IF Device.DSo.Node=0 THEN Get_Node(); END_IF
_w1 := NOT (Device.DSo.Node=0);
IF _w1 THEN Get_State(); END_IF
IF _w1 AND (Device.CanOpen.Device_State=_3SCOS.DED.DEVICE_STATE.CONFIGURED) THEN State_PreOp(); END_IF
_w2 := True;
IF _w2 THEN PDO_Units(); END_IF
IF _w2 THEN Process_Alarms(); END_IF
_w3 := Device.CanOpen.Device_State=_3SCOS.DED.DEVICE_STATE.RUNNING;
IF _w3 THEN Write_SDO(); END_IF
IF _w3 AND Device.CanOpen.Read_Once THEN Read_SDO(); END_IF
_w4 := Device.CanOpen.Device_State=_3SCOS.DED.DEVICE_STATE.RUNNING;
IF _w4 THEN
    SDO_CLK(PT := t#500ms); // Burkert_OSCAT_BASIC.CLK_PRG
END_IF
IF _w4 THEN
    AutoRead_CLK(PT := T#30s); // Burkert_OSCAT_BASIC.CLK_PRG
END_IF
IF AutoRead_CLK.Q THEN _w5 := True; END_IF
Device.CanOpen.Read_Once := _w5;
Device.PDO.NamurStatus.eNamur := SEL(Device.CanOpen.Device_State=_3SCOS.DED.DEVICE_STATE.RUNNING, eNamur107.Offline, Device.PDO.NamurStatus.eNamur);

END_FUNCTION_BLOCK

// Level_1_Devices/Burkert Library/CanOpen/CanOpen_8228
FUNCTION_BLOCK CanOpen_8228
VAR_INPUT
	Device: 	REFERENCE TO cCanOpen_8228;
	CanOpen:	REFERENCE TO _3SCOS.CANRemoteDevice_Diag;
	Conductivity_Units:eUnits:=eUnits.uS_cm;
	Temperature_Units:eUnits:=eUnits.C;
END_VAR
VAR_OUTPUT
END_VAR
VAR
	Concentration_Alarm:Burkert.Analog_Alarm_UDFB;
	Conductivity_Alarm:Burkert.Analog_Alarm_UDFB;
	Resistivity_Alarm:Burkert.Analog_Alarm_UDFB;
	TDS_Alarm:Burkert.Analog_Alarm_UDFB;
	Temp_Alarm:Burkert.Analog_Alarm_UDFB;
	
	Write_Data:Bytes_Dword;
	SDO_CLK:Burkert_OSCAT_BASIC.CLK_PRG;
	AutoRead_CLK:Burkert_OSCAT_BASIC.CLK_PRG;
	SDO_Read:CIA405.SDO_READ4;
	SDO_Write:CIA405.SDO_WRITE_DATA;

	
	
END_VAR

CanOpen_NMT();
IF Device.CanOpen.Device_State=_3SCOS.DED.DEVICE_STATE.RUNNING THEN
	AutoRead_CLK(PT:=T#60S);
	SDO_CLK(PT:=T#200MS);

	Alarms();
	IF Device.CanOpen.Read_Once THEN
		READ_SDO();
	ELSE
		Write_SDO();
	END_IF
END_IF

IF AutoRead_CLK.Q THEN
	Device.CanOpen.Read_Once:=TRUE;
END_IF
Translate();
Units();
Alarms();

Device.Ready:=(Device.Namur<2);
Device.TDS.Ready:=FPU.IsRealNumber(f:=Device.TDS.EU) AND Device.Namur<>0;
Device.Concentration.Ready:=FPU.IsRealNumber(f:=Device.Concentration.EU) AND Device.Namur<>0;
Device.Conductivity.Ready:=FPU.IsRealNumber(f:=Device.Conductivity.EU) AND Device.Namur<>0;
Device.Resistivity.Ready:=FPU.IsRealNumber(f:=Device.Resistivity.EU) AND Device.Namur<>0;
Device.Temperature.Ready:=FPU.IsRealNumber(f:=Device.Temperature.EU) AND Device.Namur<>0;

Device.DSO.StrNamur:=TO_STRING(Device.DSO.NamurNe107.eNamur);

END_FUNCTION_BLOCK

// Level_1_Devices/Burkert Library/CanOpen/CanOpen_8691
FUNCTION_BLOCK CanOpen_8691
VAR_INPUT

	LOCKOUT:BOOL;
	//Online:BOOL;
	Interlock:BOOL;
	Error_Delay_S:INT:=10;
	CanOpen:	REFERENCE TO _3SCOS.CANRemoteDevice_Diag;
	
	
	
END_VAR
VAR_OUTPUT
	Status	:INT;
	Output	:REAL;
END_VAR
VAR_IN_OUT
	Device	:cCanOpen_8691;
END_VAR
VAR

	TON_1: TON;
	TOF_0: TOF;
	R_TRIG_0: R_Trig;
	F_TRIG_0: F_Trig;

	SDO_CLK:Burkert_OSCAT_BASIC.CLK_PRG;
	AutoRead_CLK:Burkert_OSCAT_BASIC.CLK_PRG;
	SDO_Read:CIA405.SDO_READ4;
	SDO_Write:CIA405.SDO_WRITE_DATA;
	Basic_BCV:Basic_BCV_UDFB;
	
	
	CanRestart:TON;
	SetCommunicationState:_3SCOS.DED.ERROR;



END_VAR

(* body of a kind this reader does not render *)

END_FUNCTION_BLOCK

// Level_1_Devices/Burkert Library/CanOpen/CanOpen_8694
FUNCTION_BLOCK CanOpen_8694
VAR_INPUT
	CutOff:REAL:=0;
	LockOut_NC:BOOL:=TRUE;
	Permissive_NC:BOOL:=TRUE;
	Error_PCT:REAL:=10;
	Error_Delay_S:INT:=10;
	CanOpen:	REFERENCE TO _3SCOS.CANRemoteDevice_Diag;
	Device	:	REFERENCE TO cCanOpen_8694;
	
	
	
END_VAR
VAR_OUTPUT
	Status	:INT;
	Output	:REAL;
END_VAR
VAR_IN_OUT
	
END_VAR
VAR

	CanRestart:TON;

	Status_CLK:Burkert_OSCAT_BASIC.CLK_PRG;
	SDO_CLK:Burkert_OSCAT_BASIC.CLK_PRG;
	AutoRead_CLK:Burkert_OSCAT_BASIC.CLK_PRG;
	GetState_CLK:Burkert_OSCAT_BASIC.GEN_PULSE;
	SDO_Read:CIA405.SDO_READ4;
	SDO_Write:CIA405.SDO_WRITE_DATA;
	SDO_Data:ARRAY[1..4] OF BYTE;
	Write_Data:Bytes_Dword;
	
	
	Base_ACV:Basic_ACV_UDFB;
	
	SetCommunicationState:_3SCOS.DED.ERROR;
	//deiInfo:_3SCOS.DED.DEVICE_INFO;
	GetState:			CIA405.GET_STATE;
	CIA_State:			CIA405.DEVICE_STATE;
	NMT:				CIA405.NMT;
	CanState:			_3SCOS.DED.DEVICE_STATE;
	Device_State:		_3SCOS.DED.DEVICE_STATE;
	GetState_eError:	_3SCOS.DED.ERROR;
	Start_Available:BOOL;
	Ref_OK:Bool;
END_VAR

(* body of a kind this reader does not render *)

END_FUNCTION_BLOCK

// Level_1_Devices/Burkert Library/CanOpen/CanOpen_MS02
FUNCTION_BLOCK CanOpen_MS02
VAR_INPUT
	CanOpen:	REFERENCE TO _3SCOS.CANRemoteDevice_Diag;
	
END_VAR
VAR_OUTPUT
END_VAR
VAR
	SDO_CLK:Burkert_OSCAT_BASIC.CLK_PRG;
	AutoRead_CLK:Burkert_OSCAT_BASIC.CLK_PRG;
	SDO_Read:CIA405.SDO_READ4;
	SDO_Write:CIA405.SDO_WRITE_DATA;
	ALARM_0: Burkert.Analog_Alarm_UDFB;
	ALARM_1: Burkert.Analog_Alarm_UDFB;
	
END_VAR
VAR_IN_OUT
	Sensor: cCanOpen_MS02;
	
END_VAR

CanOpen_NMT();
IF Sensor.CanOpen.Device_State=_3SCOS.DED.DEVICE_STATE.RUNNING THEN
	AutoRead_CLK(PT:=T#60S);
	SDO_CLK(PT:=T#200MS);

	Alarms();
	IF Sensor.CanOpen.Read_Once THEN
		READ_SDO();
	ELSE
		Write_SDO();
	END_IF
END_IF

IF AutoRead_CLK.Q THEN
	Sensor.CanOpen.Read_Once:=TRUE;
END_IF

END_FUNCTION_BLOCK

// Level_1_Devices/Burkert Library/CanOpen/CanOpen_MS03
FUNCTION_BLOCK CanOpen_MS03
VAR_INPUT
	CanOpen:	REFERENCE TO _3SCOS.CANRemoteDevice_Diag;
	
END_VAR
VAR_OUTPUT
END_VAR
VAR
	SDO_CLK:Burkert_OSCAT_BASIC.CLK_PRG;
	AutoRead_CLK:Burkert_OSCAT_BASIC.CLK_PRG;
	SDO_Read:CIA405.SDO_READ4;
	SDO_Write:CIA405.SDO_WRITE_DATA;
	ALARM_0: Burkert.Analog_Alarm_UDFB;
	ALARM_1: Burkert.Analog_Alarm_UDFB;
	
END_VAR
VAR_IN_OUT
	Sensor: cCanOpen_MS03;
	
END_VAR

CanOpen_NMT();
IF Sensor.CanOpen.Device_State=_3SCOS.DED.DEVICE_STATE.RUNNING THEN
	AutoRead_CLK(PT:=T#60S);
	SDO_CLK(PT:=T#200MS);

	Alarms();
	IF Sensor.CanOpen.Read_Once THEN
		READ_SDO();
	ELSE
		Write_SDO();
	END_IF
END_IF

IF AutoRead_CLK.Q THEN
	Sensor.CanOpen.Read_Once:=TRUE;
END_IF

END_FUNCTION_BLOCK

// Level_1_Devices/Burkert Library/CanOpen/CanOpen_MS04
FUNCTION_BLOCK CanOpen_MS04
VAR_INPUT
	CanOpen:	REFERENCE TO _3SCOS.CANRemoteDevice_Diag;
	
END_VAR
VAR_OUTPUT
END_VAR
VAR
	SDO_CLK:Burkert_OSCAT_BASIC.CLK_PRG;
	AutoRead_CLK:Burkert_OSCAT_BASIC.CLK_PRG;
	SDO_Read:CIA405.SDO_READ4;
	SDO_Write:CIA405.SDO_WRITE_DATA;
	ALARM_0: Burkert.Analog_Alarm_UDFB;
	ALARM_1: Burkert.Analog_Alarm_UDFB;
	
END_VAR
VAR_IN_OUT
	Sensor: cCanOpen_MS04;
	
END_VAR

CanOpen_NMT();
IF Sensor.CanOpen.Device_State=_3SCOS.DED.DEVICE_STATE.RUNNING THEN
	AutoRead_CLK(PT:=T#60S);
	SDO_CLK(PT:=T#200MS);

	Alarms();
	IF Sensor.CanOpen.Read_Once THEN
		READ_SDO();
	ELSE
		Write_SDO();
	END_IF
END_IF

IF AutoRead_CLK.Q THEN
	Sensor.CanOpen.Read_Once:=TRUE;
END_IF

END_FUNCTION_BLOCK

// Level_1_Devices/Burkert Library/CanOpen/CanOpen_MS05
FUNCTION_BLOCK CanOpen_MS05
VAR_INPUT
	CanOpen:	REFERENCE TO _3SCOS.CANRemoteDevice_Diag;
	
END_VAR
VAR_OUTPUT
END_VAR
VAR
	SDO_CLK:Burkert_OSCAT_BASIC.CLK_PRG;
	AutoRead_CLK:Burkert_OSCAT_BASIC.CLK_PRG;
	SDO_Read:CIA405.SDO_READ4;
	SDO_Write:CIA405.SDO_WRITE_DATA;
	ALARM_0: Burkert.Analog_Alarm_UDFB;
	ALARM_1: Burkert.Analog_Alarm_UDFB;
	
END_VAR
VAR_IN_OUT
	Sensor: cCanOpen_MS05;
	
END_VAR

CanOpen_NMT();
IF Sensor.CanOpen.Device_State=_3SCOS.DED.DEVICE_STATE.RUNNING THEN
	AutoRead_CLK(PT:=T#60S);
	SDO_CLK(PT:=T#200MS);

	Alarms();
	IF Sensor.CanOpen.Read_Once THEN
		READ_SDO();
	ELSE
		Write_SDO();
	END_IF
END_IF

IF AutoRead_CLK.Q THEN
	Sensor.CanOpen.Read_Once:=TRUE;
END_IF

END_FUNCTION_BLOCK

// Level_1_Devices/Burkert Library/eDip/eDip_8098_CTRL
FUNCTION_BLOCK eDip_8098_CTRL
VAR_INPUT
	Device: REFERENCE TO ceDip_8098;
	Gateway: REFERENCE TO ME43_SDO;
	Node:Byte;
	Temperature_Units:eUnits:=eUnits.C;
	Flow_Units:eUnits:=eUnits.lpm;
	Volume_Units:eUnits:=eUnits.l;
END_VAR
VAR_OUTPUT
END_VAR
VAR
	Data:Bytes_Dword;
	Alarm:ARRAY[0..5] OF Burkert.Analog_Alarm_UDFB;
	Device_Valid:BOOL;
	Gateway_Valid:BOOL;
	F_trig_0:F_Trig;
	Startup_Ton:Ton;
	
	
END_VAR

Device.DSO.Node:=Node;


Device_Valid:=__ISVALIDREF(Device);
Gateway_Valid:=__ISVALIDREF(Gateway);
Device.DSO.Node:=Node;

IF  Device_Valid  THEN 
	Parse_RX();
END_IF;
StartUp_Ton(In:=Gateway_Valid AND Device_Valid ,PT:=T#1S);

IF Gateway_Valid AND StartUp_Ton.Q THEN
	Process_Alarms();
	Reset_Counters();
	Device.TCP_State:=Gateway.CommState;
	Device.strTCPstate:=TO_STRING(Device.TCP_State);
END_IF

END_FUNCTION_BLOCK

// Level_1_Devices/Burkert Library/eDip/eDip_8228_MEx3
FUNCTION_BLOCK eDip_8228_MEx3
VAR_INPUT
	Device: REFERENCE TO ceDip_8228;
	GW_Connected:BOOL;
	Node:byte;
END_VAR
VAR_OUTPUT
END_VAR
VAR
	data:Bytes_Dword;
	Concentration_Alarm:Burkert.Analog_Alarm_UDFB;
	Conductivity_Alarm:Burkert.Analog_Alarm_UDFB;
	Resistivity_Alarm:Burkert.Analog_Alarm_UDFB;
	TDS_Alarm:Burkert.Analog_Alarm_UDFB;
	Temp_Alarm:Burkert.Analog_Alarm_UDFB;
	Concentration_Native:REAL;
	Conductivity_Native:REAL;
	Resistivity_Native:REAL;
	TDS_Native:REAL;
	Temperature_Native:REAL;
	
	
END_VAR

Device.DSO.Node:=Node;
Translate();
Units();
Alarms();

Device.Ready:=(Device.Namur<2) AND GW_Connected ;
Device.TDS.Ready:=FPU.IsRealNumber(f:=Device.TDS.EU)AND GW_Connected AND Device.Namur<>0;
Device.Concentration.Ready:=FPU.IsRealNumber(f:=Device.Concentration.EU)AND GW_Connected AND Device.Namur<>0;
Device.Conductivity.Ready:=FPU.IsRealNumber(f:=Device.Conductivity.EU)AND GW_Connected AND Device.Namur<>0;
Device.Resistivity.Ready:=FPU.IsRealNumber(f:=Device.Resistivity.EU)AND GW_Connected AND Device.Namur<>0;
Device.Temperature.Ready:=FPU.IsRealNumber(f:=Device.Temperature.EU)AND GW_Connected AND Device.Namur<>0;

END_FUNCTION_BLOCK

// Level_1_Devices/Burkert Library/eDip/eDip_8312
FUNCTION_BLOCK eDip_8312
VAR_INPUT
	Device:REFERENCE TO c8312;
	GW_Connected:BOOL;
	Node:BYTE;
END_VAR
VAR_OUTPUT
END_VAR
VAR
	Alarm:Burkert.Analog_Alarm_UDFB;
	isReal:bool;
END_VAR

device.DSO.Node:=Node;
isReal:=FPU.IsRealNumber(Device.RX.EU.tReal);
IF isReal AND GW_Connected  AND device.RX.Namur.tByte[1]<>255	THEN	
	Alarm(Config:=Device.Burkert.cAlarm_Config , EU:= Device.EU, Status=> Device.Status.eStatus);
	Device.EU:=Device.RX.EU.tReal;
ELSE
	Device.Status.eStatus:=Burkert.eSensor_Status.Offline;
	Device.EU:=0;
END_IF;
Device.Ready:=isReal AND GW_Connected AND NOT(Device.Status.eStatus=Burkert.eSensor_Status.Offline);
CASE Device.RX.Namur.tByte[1] OF
	0:Device.Ready:=isReal AND GW_Connected AND NOT(Device.Status.eStatus=Burkert.eSensor_Status.Offline);
	1:	
		Device.Ready:=FALSE;
		Device.Status.eStatus:=Burkert.eSensor_Status.Fault;
	2:
		Device.Ready:=FALSE;
		Device.Status.eStatus:=Burkert.eSensor_Status.Over_Range;
	4:
		Device.Ready:=FALSE;
		Device.Status.eStatus:=Burkert.eSensor_Status.Under_Range;
END_CASE;

END_FUNCTION_BLOCK

// Level_1_Devices/Burkert Library/eDip/eDip_8412
FUNCTION_BLOCK eDip_8412
VAR_INPUT
	Device:REFERENCE TO c8412;
	GW_Connected:BOOL;
END_VAR
VAR_OUTPUT
END_VAR
VAR
	Alarm:Burkert.Analog_Alarm_UDFB;
	isReal:Bool;
END_VAR
// 8412 eDip Temperature

isReal:=FPU.IsRealNumber(Device.RX.EU.tReal);
IF isReal AND GW_Connected  AND device.RX.Namur.tByte[1]<>255	THEN	
	Alarm(Config:=Device.Burkert.cAlarm_Config , EU:= Device.EU, Status=> Device.Status.eStatus);
	Device.EU:=Device.RX.EU.tReal;
ELSE
	Device.Status.eStatus:=Burkert.eSensor_Status.Offline;
	Device.EU:=0;
END_IF;
Device.Ready:=isReal AND GW_Connected AND NOT(Device.Status.eStatus=Burkert.eSensor_Status.Offline);
CASE Device.RX.Namur.tByte[1] OF
	0:Device.Ready:=isReal AND GW_Connected AND NOT(Device.Status.eStatus=Burkert.eSensor_Status.Offline);
	1:	
		Device.Ready:=FALSE;
		Device.Status.eStatus:=Burkert.eSensor_Status.Fault;
	2:
		Device.Ready:=FALSE;
		Device.Status.eStatus:=Burkert.eSensor_Status.Over_Range;
	4:
		Device.Ready:=FALSE;
		Device.Status.eStatus:=Burkert.eSensor_Status.Under_Range;
END_CASE;

END_FUNCTION_BLOCK

// Level_1_Devices/Burkert Library/eDip/eDip_8681_UDFB
FUNCTION_BLOCK eDip_8681_UDFB
VAR_INPUT
	Feedback:WORD;
	Namur:WORD;
	Position_0:WORD;
	Position_1:WORD;
	Node:BYTE;
	Query:BOOL;
END_VAR
VAR_OUTPUT
	Setpoint:WORD;
	
END_VAR
VAR
	lcl_status: BYTE;
	tControlWord:WORD;
	F_trig_0: F_trig;
	data:Bytes_Dword;
END_VAR
VAR_IN_OUT
	Valve:eDip_8681_DUT;
	GW_Control_word:WORD;
	GW_Node:BYTE;
	
END_VAR
VAR // added by the converter: edge detectors and wires of the graphical bodies
    _w1 : BOOL;
    _w2 : ANY;
END_VAR

_w1 := True;
IF _w1 THEN ORF(); END_IF
IF _w1 THEN Cyclic(); END_IF
_w2 := (Valve.Mode=Burkert.e_8681_Modes.Auto) AND (Valve.PLC_CMD=Burkert.e_8681_Modes.Upper_Drain) OR (Valve.Mode=Burkert.e_8681_Modes.Upper_Drain);
SetPoint := SEL(_w2, SEL((Valve.Mode=Burkert.e_8681_Modes.Auto) AND (Valve.PLC_CMD=Burkert.e_8681_Modes.Lower_Drain) OR (Valve.Mode=Burkert.e_8681_Modes.Lower_Drain), SEL((Valve.Mode=Burkert.e_8681_Modes.Auto) AND (Valve.PLC_CMD=Burkert.e_8681_Modes.Open) OR (Valve.Mode=Burkert.e_8681_Modes.Open), 256, 512), 1024), 2048);
Valve.Status1 := SEL(Feedback.9, SEL(_w2, SEL(Feedback.8, SEL(Feedback.9, eB8681_Status.Unknown, eB8681_Status.Open), eB8681_Status.Blocked), eB8681_Status.Upper_Drain), eB8681_Status.Lower_Drain);

END_FUNCTION_BLOCK

// Level_1_Devices/Burkert Library/eDip/eDIP_SDO_Manager
FUNCTION_BLOCK eDIP_SDO_Manager
VAR_INPUT
	Can_SDO:ARRAY[0..9] OF cSDO_DUT;
END_VAR
VAR_OUTPUT
	ME43_SDO_Address_R1000:DWORD;
	ME43_SDO_DataLength_R1002:ARRAY[0..1]OF WORD;
	ME43_SDO_Value_R1004:ARRAY[0..1] OF WORD;
	ME43_SDO_Call_R1018:WORD;
END_VAR
VAR
	lcl_pointer: INT;
	Address:ORF;
	TON_0: ton;
	TP_0: TP;
	F_TRIG_0: F_Trig;
END_VAR
VAR // added by the converter: edge detectors and wires of the graphical bodies
    _w1, _w2, _w3, _w4, _w6, _w8, _w10, _w12 : ANY;
    _w5, _w7, _w9, _w11 : BOOL;
END_VAR

_w1 := Can_SDO[lcl_pointer].Read OR Can_SDO[lcl_pointer].Write;
IF NOT _w1 THEN _w2 := (lcl_pointer+1) MOD 10; END_IF
lcl_pointer := _w2;
IF _w1 THEN _w3 := Can_SDO[lcl_pointer].Index; END_IF
Address.SDO.Index := _w3;
IF _w1 THEN _w4 := Can_SDO[lcl_pointer].SubIndex; END_IF
Address.SDO.SubIndex := _w4;
_w5 := _w1;
IF _w5 THEN _w6 := SEL(Can_SDO[lcl_pointer].Write, Can_SDO[lcl_pointer].NodeId, Can_SDO[lcl_pointer].NodeId + 16#80); END_IF
_w7 := _w5;
IF _w7 THEN _w8 := Address.Address; END_IF
_w9 := _w7;
IF _w9 THEN _w10 := Can_SDO[lcl_pointer].Bytes; END_IF
_w11 := _w9;
IF _w11 THEN _w12 := Can_SDO[lcl_pointer].Data[1]; END_IF
TON_0(IN := _w11, PT := T#1s); // ton
TP_0(IN := TON_0.Q, PT := t#1s); // TP
F_TRIG_0(CLK := TP_0.Q); // F_Trig
Can_SDO[lcl_pointer].Read := SEL(F_TRIG_0.Q, Can_SDO[lcl_pointer].Read, False);
Can_SDO[lcl_pointer].Write := SEL(F_TRIG_0.Q, Can_SDO[lcl_pointer].Write, False);
ME43_SDO_Call_R1018 := SEL(TP_0.Q, 16#0000, 16#0100);
Address.SDO.Node := _w6;
ME43_SDO_Address_R1000 := _w8;
ME43_SDO_DataLength_R1002[1] := _w10;
ME43_SDO_Value_R1004[1] := _w12;

END_FUNCTION_BLOCK

// Level_1_Devices/Burkert Library/IoLink/s8050_UDFB
FUNCTION_BLOCK s8050_UDFB
VAR
	Data_1:Bytes_DWord;
	Data_2:Bytes_DWord;
	R_TRIG_0:R_trig;
	CLK_PRG_0: Burkert_OSCAT_BASIC.CLK_PRG;
	Requests:BYTE;
	TON_0: TON;
	
	Alarm_CND:Burkert.Analog_Alarm_UDFB;
	Alarm_Temp:Burkert.Analog_Alarm_UDFB;
	Alarm_Rate:Burkert.Analog_Alarm_UDFB;
	
END_VAR
VAR_IN_OUT
	Sensor:c8050;
	Port_Request:cIFM_AL1342_Acyclic_Request;
END_VAR

VAR_INPUT
	CommState:ModbusTCPComState;
	RX:ARRAY[0..15] OF WORD;
	Port_Response:cIFM_AL1342_Acyclic_Response;
	
	CND_Units:eUnits;
	Temp_Units:eUnits;
	Flow_Units:eUnits;
	Volume_Units:eUnits;
	
END_VAR

VAR_OUTPUT
	
END_VAR
VAR // added by the converter: edge detectors and wires of the graphical bodies
    _w1, _w3, _w7, _w9, _w13, _w15, _w19, _w21, _w23, _w25, _w27, _w29, _w31, _w33, _w35, _w36, _w38, _w41 : BOOL;
    _w2, _w4, _w5, _w6, _w8, _w10, _w11, _w12, _w14, _w16, _w17, _w18, _w20, _w22, _w24, _w26, _w28, _w30, _w32, _w34, _w37, _w39, _w40, _w42 : ANY;
END_VAR

_w1 := True;
IF _w1 THEN _w2 := RX[3]; END_IF
_w3 := _w1;
IF _w3 THEN _w4 := RX[2]; END_IF
IF _w3 THEN _w5 := Data_1.tReal; END_IF
Data_1.tWord[0] := _w2;
Data_1.tWord[1] := _w4;
_w6 := Unit_Convert(eFrom := eUnits.uS_cm, eTo := eUnits.uS_cm, Source := _w5);
Sensor.CND.EU := _w6;
_w7 := True;
IF _w7 THEN _w8 := RX[5]; END_IF
_w9 := _w7;
IF _w9 THEN _w10 := RX[4]; END_IF
IF _w9 THEN _w11 := Data_1.tReal; END_IF
Data_1.tWord[0] := _w8;
Data_1.tWord[1] := _w10;
_w12 := Unit_Convert(eFrom := eUnits.l, eTo := Volume_units, Source := _w11);
Sensor.Totalizer_1 := _w12;
_w13 := True;
IF _w13 THEN _w14 := RX[7]; END_IF
_w15 := _w13;
IF _w15 THEN _w16 := RX[6]; END_IF
IF _w15 THEN _w17 := Data_1.tReal; END_IF
Data_1.tWord[0] := _w14;
Data_1.tWord[1] := _w16;
_w18 := Unit_Convert(eFrom := eUnits.C, eTo := Temp_Units, Source := WORD_TO_REAL(RX[8]) / 10.0);
Sensor.Temp.EU := _w18;
_w19 := Sensor.HMI_Count_Reset OR Sensor.PLC_Count_Reset;
IF _w19 THEN _w20 := 16#0169; END_IF
_w21 := _w19;
IF _w21 THEN _w22 := 0; END_IF
_w23 := _w21;
IF _w23 THEN _w24 := 16#02; END_IF
_w25 := _w23;
IF _w25 THEN _w26 := 0.0; END_IF
_w27 := _w25;
IF _w27 THEN _w28 := Data_2.tByte[0]; END_IF
_w29 := _w27;
IF _w29 THEN _w30 := Data_2.tByte[1]; END_IF
_w31 := _w29;
IF _w31 THEN _w32 := Data_2.tByte[2]; END_IF
_w33 := _w31;
IF _w33 THEN _w34 := Data_2.tByte[3]; END_IF
_w35 := _w33;
IF _w35 THEN
    CLK_PRG_0(PT := t#5s); // Burkert_OSCAT_BASIC.CLK_PRG
END_IF
_w36 := _w33;
IF _w36 THEN _w37 := 4; END_IF
R_TRIG_0(CLK := CLK_PRG_0.Q AND _w36); // R_Trig
_w38 := R_TRIG_0.Q;
IF _w38 THEN _w39 := 16#FF; END_IF
IF _w38 THEN _w40 := Requests+1; END_IF
Requests := _w40;
Port_Request.Port := _w39;
Port_Request.Index := _w20;
Port_Request.SubIndex := _w22;
Port_Request.Command := _w24;
Data_2.tReal := _w26;
Port_Request.Data[3] := _w28;
Port_Request.Data[4] := _w30;
Port_Request.Data[0] := _w32;
Port_Request.Data[1] := _w34;
Port_Request.Length := _w37;
IF True THEN Status(); END_IF
TON_0(IN := (Port_request.User_ID=Port_Response.User_ID) AND (Port_Request.Index=Port_response.Index) AND Sensor.HMI_Count_Reset AND _w35, PT := T#2s); // TON
IF TON_0.Q THEN _w41 := False; END_IF
Sensor.HMI_Count_Reset := _w41;
_w42 := Unit_Convert(eFrom := eUnits.lps, eTo := Flow_Units, Source := _w17);
Sensor.Rate_1.EU := _w42;

END_FUNCTION_BLOCK

// Brite_1_UDFB
FUNCTION_BLOCK Brite_1_UDFB
VAR_INPUT
	Lower_Temperature:REAL;
	//Middle_Temperature:REAL;
	//Upper_Temperature:REAL;
	Valves_Healthy:BOOL:=TRUE;
	Sensor_Healthy:BOOL:=TRUE;
	Coolant_Healthy:BOOL:=TRUE;
	//Alarm:		REFERENCE TO Burkert.cSensor;
	//Alarm_Index:	UINT;
	//Control_Loop:REFERENCE TO cPID_DUT;
	//PID_Index:UINT;
END_VAR
VAR_OUTPUT
	Lower_ACV:REAL;
	//Middle_ACV:REAL;
	//Upper_ACV:REAL;
END_VAR
VAR
	Active_Zones: INT;
	Active_Target:REAL;
	//PID_UDFB_0: PID_UDFB;
	Vessel_Active: BOOL;
	Vessel_Error: REAL;
	R_TRIG_0: R_Trig;
	Temperature:REAL;
	TON_0: TON;
	TOF_0: TOF;
	R_TRIG_1: R_Trig;
	Loop_Reset:RS;

END_VAR
VAR_IN_OUT
	Vessel:cBrite;
	cSensor:				Burkert.cSensor;
	cAlarm_Offsets:			Burkert.cAlarm_Offsets;
	Control_Loop:		cPID_DUT;
END_VAR
VAR // added by the converter: edge detectors and wires of the graphical bodies
    _w1, _w3, _w8, _w9, _w10 : BOOL;
    _w2, _w6, _w7, _w13 : ANY;
    _w4, _w5 : REAL;
    _w11, _w12 : STRING;
END_VAR

_w1 := Vessel.Mode.eMode <> eFermenter_Modes.Off;
_w2 := (Vessel_Error>Vessel.Config.Dead_Band) OR (Vessel.Config.Dead_Band<0.1);
_w3 := _w1;
IF _w3 THEN _w4 := Temperature; END_IF
IF _w3 THEN _w5 := Active_target; END_IF
Control_Loop.Actual := _w4;
Active_Target := SEL(Vessel.Mode.eMode=eBrite_modes.ON, Temperature, Vessel.Target);
_w6 := (Vessel.Mode.eMode=eFermenter_Modes.Ferment) OR (Vessel.Mode.eMode=eFermenter_Modes.Crash);
Vessel_Active := _w6;
_w7 := SEL(_w6, 0, Temperature-Active_Target);
Vessel.Vessel_Status.Error := _w7;
Vessel_Error := _w7;
Loop_Reset(SET := Vessel.Working_Temperature_Status.eStatus=Burkert.eSensor_Status.OK, RESET1 := cSensor.Alarm_Config.Within_Norms OR (Vessel.Mode.eMode=eFermenter_Modes.Off)); // RS
R_TRIG_1(CLK := Loop_Reset.Q1); // R_Trig
TOF_0(IN := R_TRIG_1.Q, PT := T#2S); // TOF
Control_Loop.PLC_Enable := NOT TOF_0.Q AND _w2 AND _w1;
_w8 := True;
IF _w8 THEN Calculate_Zones(); END_IF
_w9 := _w8;
IF _w9 THEN Alarm_CTRL(); END_IF
IF _w9 THEN Status(); END_IF
_w10 := True;
IF _w10 THEN _w11 := TO_STRING(Vessel.Mode.eMode); END_IF
IF _w10 THEN _w12 := TO_STRING(Vessel.Status.eStatus); END_IF
Vessel.StrStatus := _w12;
Vessel.StrMode := _w11;
Vessel.Vessel_Status.Cooling_Load := Control_Loop.CV;
IF NOT Vessel_Active THEN _w13 := 0.0; END_IF
Vessel.Vessel_Status.Upper_PCT := _w13;
Vessel.Vessel_Status.Middle_PCT := _w13;
Vessel.Vessel_Status.Upper_PCT := _w13;
Lower_ACV := _w13;
Control_Loop.PLC_Target := _w5;
IF Vessel_Active THEN Active_Zones_1(); END_IF

END_FUNCTION_BLOCK

// Brite_2_UDFB
FUNCTION_BLOCK Brite_2_UDFB
VAR_INPUT
	Lower_Temperature:REAL;
	Middle_Temperature:REAL;
	//Upper_Temperature:REAL;
	Valves_Healthy:BOOL:=TRUE;
	Sensor_Healthy:BOOL:=TRUE;
	Coolant_Healthy:BOOL:=TRUE;
	//Alarm:		REFERENCE TO Burkert.cSensor;
	//Alarm_Index:	UINT;
	//Control_Loop:REFERENCE TO cPID_DUT;
	//PID_Index:UINT;
END_VAR
VAR_OUTPUT
	Lower_ACV:REAL;
	Middle_ACV:REAL;
	//Upper_ACV:REAL;
END_VAR
VAR
	Active_Zones: INT;
	Active_Target:REAL;
	//PID_UDFB_0: PID_UDFB;
	Vessel_Active: BOOL;
	Vessel_Error: REAL;
	R_TRIG_0: R_Trig;
	Temperature:REAL;
	TON_0: TON;
	TOF_0: TOF;
	R_TRIG_1: R_Trig;
	Loop_Reset:RS;

END_VAR
VAR_IN_OUT
	Vessel:cBrite;
	cSensor:				Burkert.cSensor;
	cAlarm_Offsets:			Burkert.cAlarm_Offsets;
	Control_Loop:		cPID_DUT;
END_VAR
VAR // added by the converter: edge detectors and wires of the graphical bodies
    _w1, _w3, _w8, _w9, _w10 : BOOL;
    _w2, _w6, _w7, _w13 : ANY;
    _w4, _w5 : REAL;
    _w11, _w12 : STRING;
END_VAR

IF Vessel_Active AND (Active_Zones=2) THEN Active_Zones_2(); END_IF
_w1 := Vessel.Mode.eMode <> eFermenter_Modes.Off;
_w2 := (Vessel_Error>Vessel.Config.Dead_Band) OR (Vessel.Config.Dead_Band<0.1);
_w3 := _w1;
IF _w3 THEN _w4 := Temperature; END_IF
IF _w3 THEN _w5 := Active_target; END_IF
Control_Loop.Actual := _w4;
Active_Target := SEL(Vessel.Mode.eMode=eBrite_modes.ON, Temperature, Vessel.Target);
_w6 := (Vessel.Mode.eMode=eFermenter_Modes.Ferment) OR (Vessel.Mode.eMode=eFermenter_Modes.Crash);
Vessel_Active := _w6;
_w7 := SEL(_w6, 0, Temperature-Active_Target);
Vessel.Vessel_Status.Error := _w7;
Vessel_Error := _w7;
Loop_Reset(SET := Vessel.Working_Temperature_Status.eStatus=Burkert.eSensor_Status.OK, RESET1 := cSensor.Alarm_Config.Within_Norms OR (Vessel.Mode.eMode=eFermenter_Modes.Off)); // RS
R_TRIG_1(CLK := Loop_Reset.Q1); // R_Trig
TOF_0(IN := R_TRIG_1.Q, PT := T#2S); // TOF
Control_Loop.PLC_Enable := NOT TOF_0.Q AND _w2 AND _w1;
_w8 := True;
IF _w8 THEN Calculate_Zones(); END_IF
_w9 := _w8;
IF _w9 THEN Alarm_CTRL(); END_IF
IF _w9 THEN Status(); END_IF
IF Vessel_Active AND (Active_Zones=0) THEN Active_Zones_0(); END_IF
_w10 := True;
IF _w10 THEN _w11 := TO_STRING(Vessel.Mode.eMode); END_IF
IF _w10 THEN _w12 := TO_STRING(Vessel.Status.eStatus); END_IF
Vessel.StrStatus := _w12;
Vessel.StrMode := _w11;
Vessel.Vessel_Status.Cooling_Load := Control_Loop.CV;
IF NOT Vessel_Active THEN _w13 := 0.0; END_IF
Vessel.Vessel_Status.Upper_PCT := _w13;
Vessel.Vessel_Status.Middle_PCT := _w13;
Vessel.Vessel_Status.Upper_PCT := _w13;
Lower_ACV := _w13;
Middle_ACV := _w13;
Control_Loop.PLC_Target := _w5;
IF Vessel_Active AND (Active_Zones=1) THEN Active_Zones_1(); END_IF

END_FUNCTION_BLOCK

// Brite_3_UDFB
FUNCTION_BLOCK Brite_3_UDFB
VAR_INPUT
	Lower_Temperature:REAL;
	Middle_Temperature:REAL;
	Upper_Temperature:REAL;
	Valves_Healthy:BOOL:=TRUE;
	Sensor_Healthy:BOOL:=TRUE;
	Coolant_Healthy:BOOL:=TRUE;
	//Alarm:		REFERENCE TO Burkert.cSensor;
	//Alarm_Index:	UINT;
	//Control_Loop:REFERENCE TO cPID_DUT;
	//PID_Index:UINT;
END_VAR
VAR_OUTPUT
	Lower_ACV:REAL;
	Middle_ACV:REAL;
	Upper_ACV:REAL;
END_VAR
VAR
	Active_Zones: INT;
	Active_Target:REAL;
	//PID_UDFB_0: PID_UDFB;
	Vessel_Active: BOOL;
	Vessel_Error: REAL;
	R_TRIG_0: R_Trig;
	Temperature:REAL;
	TON_0: TON;
	TOF_0: TOF;
	R_TRIG_1: R_Trig;
	Loop_Reset:RS;

	TONOF_1: Burkert_OSCAT_BASIC.TONOF;
END_VAR
VAR_IN_OUT
	Vessel:cBrite;
	cSensor:				Burkert.cSensor;
	cAlarm_Offsets:			Burkert.cAlarm_Offsets;
	Control_Loop:		cPID_DUT;
END_VAR
VAR // added by the converter: edge detectors and wires of the graphical bodies
    _w1, _w3, _w8, _w9, _w10 : BOOL;
    _w2, _w6, _w7, _w13 : ANY;
    _w4, _w5 : REAL;
    _w11, _w12 : STRING;
END_VAR

IF Vessel_Active AND (Active_Zones=2) THEN Active_Zones_2(); END_IF
IF Vessel_Active AND (Active_Zones=3) THEN Active_Zones_3(); END_IF
_w1 := Vessel.Mode.eMode <> eFermenter_Modes.Off;
_w2 := (Vessel_Error>Vessel.Config.Dead_Band) OR (Vessel.Config.Dead_Band<0.1);
_w3 := _w1;
IF _w3 THEN _w4 := Temperature; END_IF
IF _w3 THEN _w5 := Active_target; END_IF
Control_Loop.Actual := _w4;
Active_Target := SEL(Vessel.Mode.eMode=eBrite_modes.ON, Temperature, Vessel.Target);
_w6 := (Vessel.Mode.eMode=eFermenter_Modes.Ferment) OR (Vessel.Mode.eMode=eFermenter_Modes.Crash);
Vessel_Active := _w6;
_w7 := SEL(_w6, 0, Temperature-Active_Target);
Vessel.Vessel_Status.Error := _w7;
Vessel_Error := _w7;
Loop_Reset(SET := Vessel.Working_Temperature_Status.eStatus=Burkert.eSensor_Status.OK, RESET1 := cSensor.Alarm_Config.Within_Norms OR (Vessel.Mode.eMode=eFermenter_Modes.Off)); // RS
R_TRIG_1(CLK := Loop_Reset.Q1); // R_Trig
TOF_0(IN := R_TRIG_1.Q, PT := T#2S); // TOF
TONOF_1(IN := _w2, T_ON := T#15s, T_OFF := T#15s); // Burkert_OSCAT_BASIC.TONOF
Control_Loop.PLC_Enable := NOT TOF_0.Q AND TONOF_1.Q AND _w1;
_w8 := True;
IF _w8 THEN Calculate_Zones(); END_IF
_w9 := _w8;
IF _w9 THEN Alarm_CTRL(); END_IF
IF _w9 THEN Status(); END_IF
IF Vessel_Active AND (Active_Zones=0) THEN Active_Zones_0(); END_IF
_w10 := True;
IF _w10 THEN _w11 := TO_STRING(Vessel.Mode.eMode); END_IF
IF _w10 THEN _w12 := TO_STRING(Vessel.Status.eStatus); END_IF
Vessel.StrStatus := _w12;
Vessel.StrMode := _w11;
Vessel.Vessel_Status.Cooling_Load := Control_Loop.CV;
IF NOT Vessel_Active THEN _w13 := 0.0; END_IF
Vessel.Vessel_Status.Upper_PCT := _w13;
Vessel.Vessel_Status.Middle_PCT := _w13;
Vessel.Vessel_Status.Upper_PCT := _w13;
Lower_ACV := _w13;
Upper_ACV := _w13;
Middle_ACV := _w13;
Control_Loop.PLC_Target := _w5;
IF Vessel_Active AND (Active_Zones=1) THEN Active_Zones_1(); END_IF

END_FUNCTION_BLOCK

// Fermenter_1_UDFB
FUNCTION_BLOCK Fermenter_1_UDFB
VAR_INPUT
	Lower_Temperature:REAL;
	//Middle_Temperature:REAL;
	//Upper_Temperature:REAL;
	Valves_Healthy:BOOL:=TRUE;
	Sensor_Healthy:BOOL:=TRUE;
	Coolant_Healthy:BOOL:=TRUE;
	//Alarm:		REFERENCE TO Burkert.cSensor;
	//Offsets:	REFERENCE TO Burkert.cAlarm_Offsets;
	//Control_Loop:REFERENCE TO cPID_DUT;
END_VAR
VAR_OUTPUT
	Lower_ACV:REAL;
	//Middle_ACV:REAL;
	//Upper_ACV:REAL;

END_VAR
VAR
	Active_Zones: INT;
	Active_Target:REAL;
	//PID_UDFB_0: PID_UDFB;
	Vessel_Active: BOOL;
	Vessel_Error: REAL;
	R_TRIG_0: R_Trig;
	Temperature:REAL;
	TON_0: TON;
	TOF_0: TOF;
	R_TRIG_1: R_Trig;
	Loop_Reset:RS;
	Init_Complete:BOOL:=FALSE;

	TONOF_0: Burkert_OSCAT_BASIC.TONOF;
END_VAR
VAR_IN_OUT
	Vessel:				cFermenter_DUT;
	cSensor:				Burkert.cSensor;
	cAlarm_Offsets:			Burkert.cAlarm_Offsets;
	Control_Loop:		cPID_DUT;
END_VAR

IF NOT Init_Complete THEN Init(); END_IF
IF Init_Complete THEN Main(); END_IF

END_FUNCTION_BLOCK

// Fermenter_2_UDFB
FUNCTION_BLOCK Fermenter_2_UDFB
VAR_INPUT
	Lower_Temperature:REAL;
	Middle_Temperature:REAL;
	//Upper_Temperature:REAL;
	Valves_Healthy:BOOL:=TRUE;
	Sensor_Healthy:BOOL:=TRUE;
	Coolant_Healthy:BOOL:=TRUE;
	//Alarm:		REFERENCE TO Burkert.cSensor;
	//Alarm_Index:	UINT;
	//Control_Loop:REFERENCE TO cPID_DUT;
	//PID_Index:UINT;
END_VAR
VAR_OUTPUT
	Lower_ACV:REAL;
	Middle_ACV:REAL;
	//Upper_ACV:REAL;
END_VAR
VAR
	Active_Zones: INT;
	Active_Target:REAL;
	//PID_UDFB_0: PID_UDFB;
	Vessel_Active: BOOL;
	Vessel_Error: REAL;
	R_TRIG_0: R_Trig;
	Temperature:REAL;
	TON_0: TON;
	TOF_0: TOF;
	R_TRIG_1: R_Trig;
	Loop_Reset:RS;

END_VAR
VAR_IN_OUT
	Vessel:					cFermenter_DUT;
	cSensor:				Burkert.cSensor;
	cAlarm_Offsets:			Burkert.cAlarm_Offsets;
	Control_Loop:			cPID_DUT;
END_VAR
VAR // added by the converter: edge detectors and wires of the graphical bodies
    _w1, _w2, _w4, _w9, _w10 : BOOL;
    _w3, _w7, _w8, _w13 : ANY;
    _w5, _w6 : REAL;
    _w11, _w12 : STRING;
END_VAR

IF Vessel_Active AND (Active_Zones=2) THEN Active_Zones_2(); END_IF
_w1 := True;
IF _w1 THEN Calculate_Zones(); END_IF
_w2 := Vessel.Mode.eMode <> eFermenter_Modes.Off;
_w3 := (Vessel_Error>Vessel.Config.Dead_Band) OR (Vessel.Config.Dead_Band<0.1);
_w4 := _w2;
IF _w4 THEN _w5 := Temperature; END_IF
IF _w4 THEN _w6 := Active_target; END_IF
Control_Loop.Actual := _w5;
Active_Target := SEL(Vessel.Mode.eMode=eFermenter_Modes.Crash, Vessel.Fermentation_Target, Vessel.Crash_Target);
_w7 := (Vessel.Mode.eMode=eFermenter_Modes.Ferment) OR (Vessel.Mode.eMode=eFermenter_Modes.Crash);
Vessel_Active := _w7;
_w8 := SEL(_w7, 0, Temperature-Active_Target);
Vessel.Vessel_Status.Error := _w8;
Vessel_Error := _w8;
Loop_Reset(SET := Vessel.Working_Temperature_Status.eStatus=Burkert.eSensor_Status.OK, RESET1 := NOT cSensor.Alarm_Config.Within_Norms OR (Vessel.Mode.eMode=eFermenter_Modes.Off)); // RS
R_TRIG_1(CLK := Loop_Reset.Q1); // R_Trig
TOF_0(IN := R_TRIG_1.Q, PT := T#2S); // TOF
Control_Loop.PLC_Enable := NOT TOF_0.Q AND _w3 AND _w2;
_w9 := _w1;
IF _w9 THEN Alarm_CTRL(); END_IF
_w10 := True;
IF _w10 THEN _w11 := TO_STRING(Vessel.Mode.eMode); END_IF
IF _w10 THEN _w12 := TO_STRING(Vessel.Status.eStatus); END_IF
Vessel.StrStatus := _w12;
Vessel.StrMode := _w11;
IF _w9 THEN Status(); END_IF
Vessel.Vessel_Status.Cooling_Load := Control_Loop.cv;
IF Vessel_Active AND (Active_Zones=0) THEN Active_Zones_0(); END_IF
IF NOT Vessel_Active THEN _w13 := 0.0; END_IF
Vessel.Vessel_Status.Lower_PCT := _w13;
Vessel.Vessel_Status.Middle_PCT := _w13;
Vessel.Vessel_Status.Upper_PCT := _w13;
Lower_ACV := _w13;
Middle_ACV := _w13;
Control_Loop.PLC_Target := _w6;
IF Vessel_Active AND (Active_Zones=1) THEN Active_Zones_1(); END_IF

END_FUNCTION_BLOCK

// Fermenter_3_UDFB
FUNCTION_BLOCK Fermenter_3_UDFB
VAR_INPUT
	Lower_Temperature:REAL;
	Middle_Temperature:REAL;
	Upper_Temperature:REAL;
	Valves_Healthy:BOOL:=TRUE;
	Sensor_Healthy:BOOL:=TRUE;
	Coolant_Healthy:BOOL:=TRUE;
		//Alarm:		REFERENCE TO Burkert.cSensor;
	//Alarm_Index:	UINT;
	//Control_Loop:REFERENCE TO cPID_DUT;
	//PID_Index:UINT;
END_VAR
VAR_OUTPUT
	Lower_ACV:REAL;
	Middle_ACV:REAL;
	Upper_ACV:REAL;
END_VAR
VAR
	Active_Zones: INT;
	Active_Target:REAL;
	//PID_UDFB_0: PID_UDFB;
	Vessel_Active: BOOL;
	Vessel_Error: REAL;
	R_TRIG_0: R_Trig;
	Temperature:REAL;
	TON_0: TON;
	TOF_0: TOF;
	R_TRIG_1: R_Trig;
	Loop_Reset:RS;
END_VAR
VAR_IN_OUT
	Vessel:				cFermenter_DUT;
	cSensor:				Burkert.cSensor;
	cAlarm_Offsets:			Burkert.cAlarm_Offsets;
	Control_Loop:		cPID_DUT;
END_VAR
VAR // added by the converter: edge detectors and wires of the graphical bodies
    _w1, _w2, _w4, _w9, _w10 : BOOL;
    _w3, _w7, _w8, _w13 : ANY;
    _w5, _w6 : REAL;
    _w11, _w12 : STRING;
END_VAR

IF Vessel_Active AND (Active_Zones=2) THEN Active_Zones_2(); END_IF
IF Vessel_Active AND (Active_Zones=3) THEN Active_Zones_3(); END_IF
_w1 := True;
IF _w1 THEN Calculate_Zones(); END_IF
_w2 := Vessel.Mode.eMode <> eFermenter_Modes.Off;
_w3 := (Vessel_Error>Vessel.Config.Dead_Band) OR (Vessel.Config.Dead_Band<0.1);
_w4 := _w2;
IF _w4 THEN _w5 := Temperature; END_IF
IF _w4 THEN _w6 := Active_target; END_IF
Control_Loop.Actual := _w5;
Active_Target := SEL(Vessel.Mode.eMode=eFermenter_Modes.Crash, Vessel.Fermentation_Target, Vessel.Crash_Target);
_w7 := (Vessel.Mode.eMode=eFermenter_Modes.Ferment) OR (Vessel.Mode.eMode=eFermenter_Modes.Crash);
Vessel_Active := _w7;
_w8 := SEL(_w7, 0, Temperature-Active_Target);
Vessel.Vessel_Status.Error := _w8;
Vessel_Error := _w8;
Loop_Reset(SET := Vessel.Working_Temperature_Status.eStatus=Burkert.eSensor_Status.OK, RESET1 := NOT cSensor.Alarm_Config.Within_Norms OR (Vessel.Mode.eMode=eFermenter_Modes.Off)); // RS
R_TRIG_1(CLK := Loop_Reset.Q1); // R_Trig
TOF_0(IN := R_TRIG_1.Q, PT := T#2S); // TOF
Control_Loop.PLC_Enable := NOT TOF_0.Q AND _w3 AND _w2;
_w9 := _w1;
IF _w9 THEN Alarm_CTRL(); END_IF
_w10 := True;
IF _w10 THEN _w11 := TO_STRING(Vessel.Mode.eMode); END_IF
IF _w10 THEN _w12 := TO_STRING(Vessel.Status.eStatus); END_IF
Vessel.StrStatus := _w12;
Vessel.StrMode := _w11;
IF _w9 THEN Status(); END_IF
Vessel.Vessel_Status.Cooling_Load := Control_Loop.CV;
IF NOT Vessel_Active THEN _w13 := 0.0; END_IF
Vessel.Vessel_Status.Lower_PCT := _w13;
Vessel.Vessel_Status.Middle_PCT := _w13;
Vessel.Vessel_Status.Upper_PCT := _w13;
Lower_ACV := _w13;
Upper_ACV := _w13;
Middle_ACV := _w13;
Control_Loop.PLC_Target := _w6;
IF Vessel_Active AND (Active_Zones=1) THEN Active_Zones_1(); END_IF

END_FUNCTION_BLOCK

// CLT
PROGRAM CLT
VAR
	
	Local_Task:eCLT_Task;
	SW_Valid:BOOL;
	SW_Ton:TON;
	Dummy_SW:cBatch_Transfer;
	
END_VAR
VAR_OUTPUT
	Init:BOOL:=FALSE;
END_VAR

VAR_INPUT
	Config:		REFERENCE TO CLT_DUT;
	
	Tank_LSHH: REFERENCE TO DI_DUT;
	Pump_Intake_LS	:REFERENCE TO DI_DUT;
	
	Tank_Level:		REFERENCE TO Burkert.cAIT;
	Temperature		:REFERENCE TO Burkert.cAIT;
	HTX_Discharge_TT	:REFERENCE TO Burkert.cAIT;
	Discharge_Pressure	:REFERENCE TO Burkert.cAIT;
	
	Recirc_FIT			:REFERENCE TO Burkert.cFIT;
	KT_FIT				:REFERENCE TO Burkert.cFIT;
	
	Recirc_ACV			:REFERENCE TO Burkert.cACV;
	Glycol_ACV			:REFERENCE TO Burkert.cACV;
	
	Fill_BCV			:REFERENCE TO Burkert.cBCV;
	
	PID_Recirc			:REFERENCE TO cPID_DUT;
	PID_Temp			:REFERENCE TO cPID_DUT;
	
	Pump:REFERENCE TO Burkert.VFD_Control;
	
	//External_Demand:Real;
END_VAR

IF NOT(Init) THEN
	do_INIT();
ELSE
	CLT_PID_CTRL();
	CLT_ACV_CTRL();
	CLT_BCV_CTRL();
	CLT_VFD_CTRL();
	Aux();
	CLT_Task_Manager();
	
END_IF

END_PROGRAM

// Grain_Room_Hopper_1Conveyor
PROGRAM Grain_Room_Hopper_1Conveyor
VAR
	
	Local_Task:eKT_Task;
	Task_Ton:TON;
	tHopper_Weight:REAL;
	Pulse_5s:Burkert_OSCAT_BASIC.CLK_PRG;
	Hopper_Empty_TON:TON;
END_VAR

VAR_IN_OUT
	Config		: GR_DUT;
	Conveyor_2	: Burkert.VFD_Control;
	
	Hopper_Gate_Valve	:Burkert.cBCV;
	Hydrator_Gate_Valve	: Burkert.cBCV;
	
	Scale		: Burkert.cAIT;
	
	MM_Task:eMM_Task;
	MM_Status:eMM_Status;
	MM_Task_ETA:UINT;
	Strike_Valve_Status:Burkert.eBCV_Status;
END_VAR

VAR_OUTPUT
	Init:BOOL;
END_VAR

IF NOT(Init) THEN
	Do_INIT();
ELSE
	Pulse_5s(PT:=T#5S);
	Hopper_Empty_TON(PT:=T#15S);
	AUX();
	Task_Manager();
	GR_BCV_CTRL();
	GR_VFD_CTRL();
	

END_IF;

END_PROGRAM

// HLT_2Pump_2Mix
PROGRAM HLT_2Pump_2Mix
VAR
	RAMP_REAL_0: RAMP_REAL;
	TON_0: TON;
	Task_Ton:TON;
	SW_Ton:TON;
	
	Current_Task:eHLT_Task;
	Current_Mode:eHLT_Modes;
	SW_Valid:BOOL:=FALSE;
	
	Dummy_SW:cBatch_Transfer;
	Dummy_BCV:Burkert.cBCV;
END_VAR
VAR_OUTPUT
	Init:BOOL;
END_VAR
VAR_INPUT
	Config: REFERENCE TO Config_DUT;
	RTC:REFERENCE TO SysTimeDate;
	Day_Seconds:UDINT;
	
	Strike_HW:REFERENCE TO Burkert.cACV;
	Strike_CW:REFERENCE TO Burkert.cACV;
	Sparge_HW:REFERENCE TO Burkert.cACV;
	Sparge_CW:REFERENCE TO Burkert.cACV;
	HTX_Outlet_ACV:REFERENCE TO Burkert.cACV;
	HTX_Steam:REFERENCE TO Burkert.cACV;
	
	
	Mix_Pump:REFERENCE TO Burkert.VFD_Control;
	Recirc_Pump:REFERENCE TO Burkert.VFD_Control;
	
	
	
	Strike_FIT:REFERENCE TO Burkert.cFIT;
	Sparge_FIT:REFERENCE TO Burkert.cFIT;
	HTX_FIT:REFERENCE TO Burkert.cFIT;
	
	CW_Fill:REFERENCE TO Burkert.cBCV;
	Recirc_To_HTX:REFERENCE TO Burkert.cBCV;
	SprayBall:REFERENCE TO Burkert.cBCV;
	SW_Main_BCV:REFERENCE TO Burkert.cBCV;
	
	
	PID_HTX:REFERENCE TO PID_DUT;
	PID_Recirc:REFERENCE TO PID_DUT;
	
	Temperature:REFERENCE TO Burkert.cAIT;
	Strike_TT:REFERENCE TO Burkert.cAIT;
	Sparge_TT:REFERENCE TO Burkert.cAIT;
	HTX_Outlet_TT:REFERENCE TO Burkert.cAIT;
	HTX_Inlet_TT:REFERENCE TO Burkert.cAIT;
	
	Mix_Pump_Pressure:REFERENCE TO Burkert.cAIT;
	Recirc_Pressure:REFERENCE TO Burkert.cAIT;
	Level:REFERENCE TO Burkert.cAIT;
	
	Pump_Intake_LSLL:REFERENCE TO DI_DUT;
	Tank_LSHH:REFERENCE TO DI_DUT;
END_VAR

IF NOT(Init) THEN
	Init_Block();
ELSE
	Aux();
	Alarms();
	HLT_Valves();
	PID();
	VFD();
	Status();
	Task_Manager();
	Tasks();
	
	
	IF SW_Valid THEN
		Service_Water_CTRL();
	END_IF;
	
	
	
END_IF;

END_PROGRAM

// HLT_2Pump_2Mix_OLD
PROGRAM HLT_2Pump_2Mix_OLD
VAR
	R_TRIG_0: R_trig;
	R_TRIG_3: R_trig;
	R_TRIG_1: R_trig;
	R_TRIG_2: R_trig;
	Alarm_Manager_0: Alarm_Manager;
	//Service_Water_Manager_0: Service_Water_Manager;
	HLT_Valve_Manager_0: HLT_Valve_Manager;
	HLT_PID_Manager_0: HLT_PID_MANAGER;
	HLT_Status_Manager_0: HLT_STATUS_MANAGER;
	HLT_VFD_Ctrl_0: HLT_VFD_Ctrl;
	HLT_Task_Manager_0: HLT_Task_Manager;
	HLT_Tasks_0: HLT_Tasks;
	Service_Water_0: Service_Water;

	F_TRIG_0: F_Trig;
END_VAR
VAR_INPUT
	Config: REFERENCE TO Config_DUT;
	RTC:REFERENCE TO SysTimeDate;
	Day_Seconds:UDINT;
	
	Strike_HW:REFERENCE TO ACV_DUT;
	Strike_CW:REFERENCE TO ACV_DUT;
	Sparge_HW:REFERENCE TO ACV_DUT;
	Sparge_CW:REFERENCE TO ACV_DUT;
	HTX_Outlet_ACV:REFERENCE TO ACV_DUT;
	HTX_Steam:REFERENCE TO ACV_DUT;
	
	
	Mix_Pump:REFERENCE TO Burkert.VFD_Control;
	Recirc_Pump:REFERENCE TO Burkert.VFD_Control;
	
	
	
	Strike_FIT:REFERENCE TO FIT_DUT;
	Sparge_FIT:REFERENCE TO FIT_DUT;
	HTX_FIT:REFERENCE TO FIT_DUT;
	Service_Water_FIT:REFERENCE TO FIT_DUT;
	
	CW_Fill:REFERENCE TO BCV_DUT;
	Recirc_To_HTX:REFERENCE TO BCV_DUT;
	SprayBall:REFERENCE TO BCV_DUT;
	
	
	PID_HTX:REFERENCE TO PID_DUT;
	PID_Recirc:REFERENCE TO PID_DUT;
	
	Temperature:REFERENCE TO AIT_DUT;
	Strike_TT:REFERENCE TO AIT_DUT;
	Sparge_TT:REFERENCE TO AIT_DUT;
	HTX_Outlet_TT:REFERENCE TO AIT_DUT;
	HTX_Inlet_TT:REFERENCE TO AIT_DUT;
	
	Mix_Pump_Pressure:REFERENCE TO AIT_DUT;
	Recirc_Pressure:REFERENCE TO Ait_DUT;
	Level:REFERENCE TO AIT_DUT;
	
	Pump_Intake_LSLL:REFERENCE TO DI_DUT;
	Tank_LSHH:REFERENCE TO DI_DUT;
END_VAR
VAR // added by the converter: edge detectors and wires of the graphical bodies
    _w1, _w8, _w9, _w10, _w11, _w12, _w13, _w15, _w17, _w19, _w21, _w24, _w26, _w27, _w29, _w30 : ANY;
    _w2, _w3, _w4, _w5, _w6, _w7, _w14, _w16, _w18, _w20, _w22, _w23, _w25, _w28 : BOOL;
END_VAR

